//{attribute 'qualified_only'}
{attribute 'strict'}
TYPE E_DataSets :
(
	DataSet1 := 10,
	DataSet2 := 11,
	DataSet3 := 12
);
END_TYPE

(* stored: Version 1.1.0.1, ProductVersion 3.1.4024.4
   DUT E_DataSets: Id {9332fdc6-cb97-4f47-8d17-d6f2bd8d0944} *)
